(********************* G.D S.p.A. - Technical Department ***********************************
This program has been generated automatically from Application Designer DE&F
********************************************************************************************)
PROGRAM dbg_csp_case_fc_ls_upper_sensors
VAR
  flap_chksect_shd : check_section_shadow;
  flap_di_shd : digital_input_shadow;
END_VAR

_objects_manager();

IF	g_application_status <> APPLICATION_STATUS_RUNNING
THEN
	RETURN;
END_IF

CASE process_get_mode(CONVERSION_this := dbg_root.prc) OF
	MODE_ABSENT,
	MODE_INACTIVE:
		RETURN;
	MODE_TEST:
		RETURN;
END_CASE

ACTION _objects_manager:
IF	objects_initialization()
THEN
	check_section_shadow_init(
		sim_mode:= SHADOW_SIMULATION_MODE_AUTOMATIC, 
		father:= csp_case_fc_ls_upper_sensors.flap_chksect, 
		process:= dbg_root.prc, 
		CONVERSION_this:= flap_chksect_shd);

	digital_input_shadow_init(
		sim_mode:= SHADOW_SIMULATION_MODE_AUTOMATIC, 
		father:= csp_case_fc_ls_upper_sensors.flap_di, 
		process:= dbg_root.prc, 
		CONVERSION_this:= flap_di_shd);

	RETURN;
END_IF

IF	objects_running()
THEN
	digital_input_shadow_cycle(flap_di_shd);
END_IF
END_ACTION

END_PROGRAM

(* stored: Version 1.1.0.1, ProductVersion 3.1.4022.12
   POU dbg_csp_case_fc_ls_upper_sensors: Id {098f6f8e-e312-4087-a757-50f7e8321834}, SpecialFunc None
   Action _objects_manager: Id {20c7f890-d314-487a-af76-0f1cd3abe076} *)
